(****************************************************************************************)
(*							Beckhoff Automation Poland									*)
(*								arrBOOL8_TO_BYTE v1.0									*)
(*									15.02.2010											*)
(*		Funkcja tworząca zmienną typu BYTE z tablicy 8 zmiennych typu BOOL				*)
(*______________________________________________________________________________________*)
FUNCTION arrBOOL8_TO_BYTE : BYTE
VAR_INPUT
	aBool8 : ARRAY [0..7] OF BOOL;
END_VAR

arrBOOL8_TO_BYTE.0 := aBool8[0];
arrBOOL8_TO_BYTE.1 := aBool8[1];
arrBOOL8_TO_BYTE.2 := aBool8[2];
arrBOOL8_TO_BYTE.3 := aBool8[3];
arrBOOL8_TO_BYTE.4 := aBool8[4];
arrBOOL8_TO_BYTE.5 := aBool8[5];
arrBOOL8_TO_BYTE.6 := aBool8[6];
arrBOOL8_TO_BYTE.7 := aBool8[7];

END_FUNCTION

(* stored: Version 1.1.0.1, ProductVersion 3.1.4026.13, FileIdentifier c1f4889c5100370d9ca6e7f100455fb5afc8dcee, FileSignature 8a15f9e7778c8ba296c9d090d95fd31f74abb947e07672d4275f95e4c0185594d10abc77b5029007dd53091e8126890065f7c3fcb443d6ca16e8c99950349b900dd38f00224ebd6037ebb1acbd7e351dd6246af0b6c76159d0185b49926e58646e1719cf0072941044a349b3c68128f5ae930b990c87706ab8c5934889e956d9c985450860b113de1b57c7805c06f6fb3db61d1c6cab0e9e87b64507e885bcf24cd3c5647b8b3b87298bc1af7a7b650b6ad90efc885eebe6a6a932d561bfe5611e92d2a1991525fca51e2f32a4265479e5f7e2f4c890ba9fcfafdd1250caa31684cfd84a2482043f5aefab1f4cd0d17467c163f9442d7704dd1af4d85844c18b
   POU arrBOOL8_TO_BYTE: Id {d2c9bd6d-5fed-4c33-a21c-5c24686c4625}, SpecialFunc None *)
